(* CoDeSys 2.3.9.50 project: 5B.pr6 *)
(* Libraries: STANDARD.LB6 5.6.98 12:03:02 *)

(* POU MAIN, LD *)
PROGRAM MAIN
VAR
	Start AT %IX0.0: BOOL;
	PackCans6 AT %IX0.1: BOOL;
	PackCans8 AT %IX0.2: BOOL;
	PackCans12 AT %IX0.3: BOOL;
	C1: CTU;
	C2: CTU;
	C3: CTU;
	Multiply AT %IX0.4: BOOL;
	A: INT;
	B: INT;
	C: INT;
	Total AT %IX0.5: BOOL;
	TotalCans: INT;
	Reset AT %IX0.7: BOOL;
END_VAR
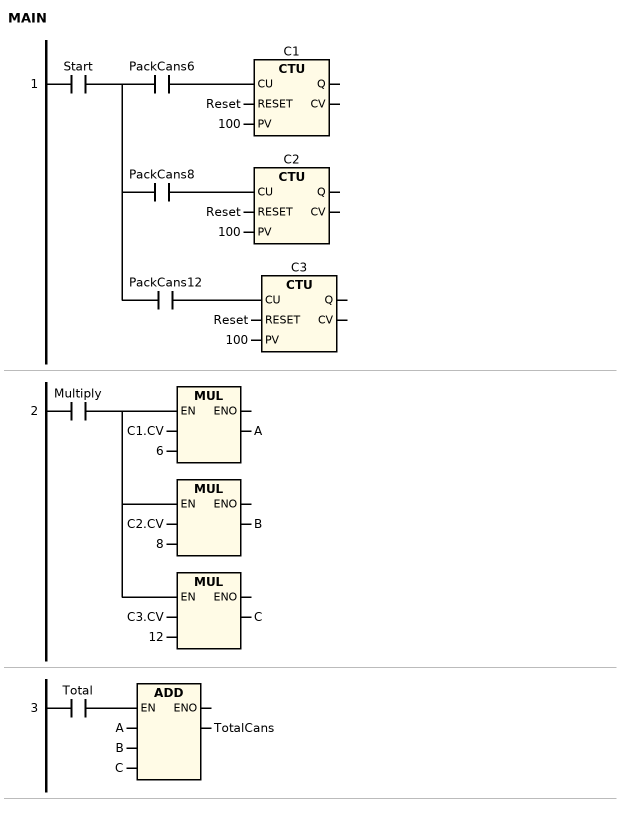
_LD_ (* Ladder Diagram *)
NETWORK 1
	[Start] - { [PackCans6] - C1:CTU(CU: *, RESET: Reset, PV: 100) | [PackCans8] - C2:CTU(CU: *, RESET: Reset, PV: 100) | [PackCans12] - C3:CTU(CU: *, RESET: Reset, PV: 100) }
NETWORK 2
	[Multiply]
		EN --- MUL(C1.CV, 6) => A
		EN --- MUL(C2.CV, 8) => B
		EN --- MUL(C3.CV, 12) => C
NETWORK 3
	[Total]
		EN --- ADD(A, B, C) => TotalCans
_END_LD_
(* the same logic as Structured Text *)
(* Network 1 *)
C1(CU := Start AND PackCans6, RESET := Reset, PV := 100);
C2(CU := Start AND PackCans8, RESET := Reset, PV := 100);
C3(CU := Start AND PackCans12, RESET := Reset, PV := 100);
(* Network 2 *)
IF Multiply THEN
	A := C1.CV * 6;
	B := C2.CV * 8;
	C := C3.CV * 12;
END_IF;
(* Network 3 *)
IF Total THEN
	TotalCans := A + B + C;
END_IF;
END_PROGRAM
